Staubli VAL3: OnF1.pgx

program OnF1()
begin
  if nType==1
    call SetFrame(sItem)
    popUpMsg("选择坐标系："+sItem)
  endIf
end
